SYSTEM Scenario_1
  (* Version 1.0, 2025-08-19, DEVIASH *)
  APPLICATION Scenario_1App (* VDMA *)
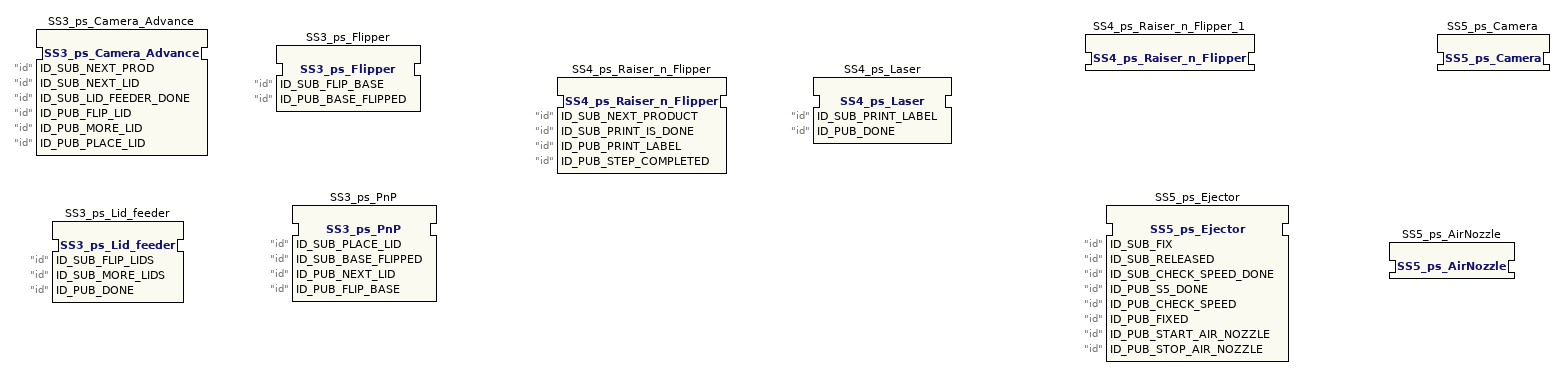
    (* Group S3_Capping_Station: Puting cap on the spinner *)
    (* Group S4_Laser_Print: Printing label on spinner using Laser *)
    (* Group S5_Quality: Speed and label quality check *)
    FBS
      SS3_ps_PnP : SS3_ps_PnP(ID_SUB_PLACE_LID := "id", ID_SUB_BASE_FLIPPED := "id", ID_PUB_NEXT_LID := "id", ID_PUB_FLIP_BASE := "id"); {SET_ATTRIBUTE(GroupName, S3_Capping_Station)}
      SS3_ps_Flipper : SS3_ps_Flipper(ID_SUB_FLIP_BASE := "id", ID_PUB_BASE_FLIPPED := "id"); {SET_ATTRIBUTE(GroupName, S3_Capping_Station)}
      SS3_ps_Lid_feeder : SS3_ps_Lid_feeder(ID_SUB_FLIP_LIDS := "id", ID_SUB_MORE_LIDS := "id", ID_PUB_DONE := "id"); {SET_ATTRIBUTE(GroupName, S3_Capping_Station)}
      SS3_ps_Camera_Advance : SS3_ps_Camera_Advance(ID_SUB_NEXT_PROD := "id", ID_SUB_NEXT_LID := "id", ID_SUB_LID_FEEDER_DONE := "id", ID_PUB_FLIP_LID := "id", ID_PUB_MORE_LID := "id", ID_PUB_PLACE_LID := "id"); {SET_ATTRIBUTE(GroupName, S3_Capping_Station)}
      SS4_ps_Raiser_n_Flipper : SS4_ps_Raiser_n_Flipper(ID_SUB_NEXT_PRODUCT := "id", ID_SUB_PRINT_IS_DONE := "id", ID_PUB_PRINT_LABEL := "id", ID_PUB_STEP_COMPLETED := "id"); {SET_ATTRIBUTE(GroupName, S4_Laser_Print)}
      SS4_ps_Laser : SS4_ps_Laser(ID_SUB_PRINT_LABEL := "id", ID_PUB_DONE := "id"); {SET_ATTRIBUTE(GroupName, S4_Laser_Print)}
      SS5_ps_Ejector : SS5_ps_Ejector(ID_SUB_FIX := "id", ID_SUB_RELEASED := "id", ID_SUB_CHECK_SPEED_DONE := "id", ID_PUB_S5_DONE := "id", ID_PUB_CHECK_SPEED := "id", ID_PUB_FIXED := "id", ID_PUB_START_AIR_NOZZLE := "id", ID_PUB_STOP_AIR_NOZZLE := "id"); {SET_ATTRIBUTE(GroupName, S5_Quality)}
      SS5_ps_AirNozzle : SS5_ps_AirNozzle; {SET_ATTRIBUTE(GroupName, S5_Quality)}
      SS4_ps_Raiser_n_Flipper_1 : SS4_ps_Raiser_n_Flipper; {SET_ATTRIBUTE(GroupName, S5_Quality)}
      SS5_ps_Camera : SS5_ps_Camera; {SET_ATTRIBUTE(GroupName, S5_Quality)}
    END_FBS
  END_APPLICATION
  APPLICATION Scenario_1_with_split_S5App
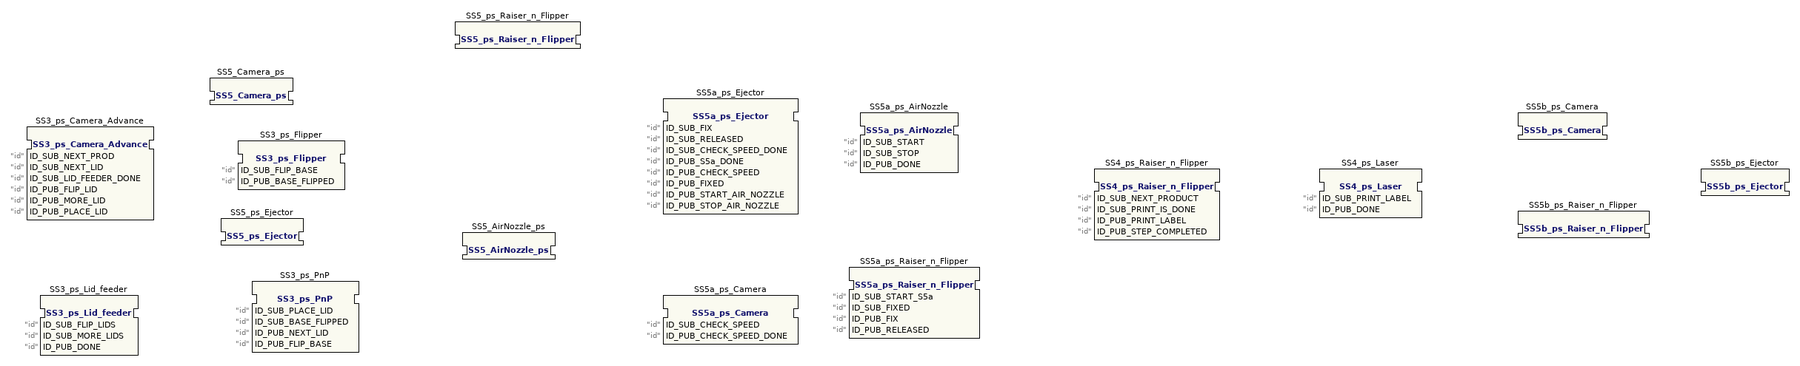
    (* Group S4_Laser_Print: Printing label on spinner using Laser *)
    (* Group S3_Capping_Station: Puting cap on the spinner *)
    (* Group S5a: Speed Quality Check *)
    (* Group S5b: Label Quality Check *)
    FBS
      SS4_ps_Raiser_n_Flipper : SS4_ps_Raiser_n_Flipper(ID_SUB_NEXT_PRODUCT := "id", ID_SUB_PRINT_IS_DONE := "id", ID_PUB_PRINT_LABEL := "id", ID_PUB_STEP_COMPLETED := "id"); {SET_ATTRIBUTE(GroupName, S4_Laser_Print)}
      SS4_ps_Laser : SS4_ps_Laser(ID_SUB_PRINT_LABEL := "id", ID_PUB_DONE := "id"); {SET_ATTRIBUTE(GroupName, S4_Laser_Print)}
      SS3_ps_PnP : SS3_ps_PnP(ID_SUB_PLACE_LID := "id", ID_SUB_BASE_FLIPPED := "id", ID_PUB_NEXT_LID := "id", ID_PUB_FLIP_BASE := "id"); {SET_ATTRIBUTE(GroupName, S3_Capping_Station)}
      SS3_ps_Flipper : SS3_ps_Flipper(ID_SUB_FLIP_BASE := "id", ID_PUB_BASE_FLIPPED := "id"); {SET_ATTRIBUTE(GroupName, S3_Capping_Station)}
      SS3_ps_Lid_feeder : SS3_ps_Lid_feeder(ID_SUB_FLIP_LIDS := "id", ID_SUB_MORE_LIDS := "id", ID_PUB_DONE := "id"); {SET_ATTRIBUTE(GroupName, S3_Capping_Station)}
      SS3_ps_Camera_Advance : SS3_ps_Camera_Advance(ID_SUB_NEXT_PROD := "id", ID_SUB_NEXT_LID := "id", ID_SUB_LID_FEEDER_DONE := "id", ID_PUB_FLIP_LID := "id", ID_PUB_MORE_LID := "id", ID_PUB_PLACE_LID := "id"); {SET_ATTRIBUTE(GroupName, S3_Capping_Station)}
      SS5_AirNozzle_ps : SS5_AirNozzle_ps; {SET_ATTRIBUTE(GroupName, S5_Quality)}
      SS5_Camera_ps : SS5_Camera_ps; {SET_ATTRIBUTE(GroupName, S5_Quality)}
      SS5_ps_Ejector : SS5_ps_Ejector; {SET_ATTRIBUTE(GroupName, S5_Quality)}
      SS5_ps_Raiser_n_Flipper : SS5_ps_Raiser_n_Flipper; {SET_ATTRIBUTE(GroupName, S5_Quality)}
      SS5a_ps_AirNozzle : SS5a_ps_AirNozzle(ID_SUB_START := "id", ID_SUB_STOP := "id", ID_PUB_DONE := "id"); {SET_ATTRIBUTE(GroupName, S5a)}
      SS5a_ps_Camera : SS5a_ps_Camera(ID_SUB_CHECK_SPEED := "id", ID_PUB_CHECK_SPEED_DONE := "id"); {SET_ATTRIBUTE(GroupName, S5a)}
      SS5a_ps_Ejector : SS5a_ps_Ejector(ID_SUB_FIX := "id", ID_SUB_RELEASED := "id", ID_SUB_CHECK_SPEED_DONE := "id", ID_PUB_S5a_DONE := "id", ID_PUB_CHECK_SPEED := "id", ID_PUB_FIXED := "id", ID_PUB_START_AIR_NOZZLE := "id", ID_PUB_STOP_AIR_NOZZLE := "id"); {SET_ATTRIBUTE(GroupName, S5a)}
      SS5b_ps_Camera : SS5b_ps_Camera; {SET_ATTRIBUTE(GroupName, S5b)}
      SS5b_ps_Ejector : SS5b_ps_Ejector; {SET_ATTRIBUTE(GroupName, S5b)}
      SS5b_ps_Raiser_n_Flipper : SS5b_ps_Raiser_n_Flipper; {SET_ATTRIBUTE(GroupName, S5b)}
      SS5a_ps_Raiser_n_Flipper : SS5a_ps_Raiser_n_Flipper(ID_SUB_START_S5a := "id", ID_SUB_FIXED := "id", ID_PUB_FIX := "id", ID_PUB_RELEASED := "id"); {SET_ATTRIBUTE(GroupName, S5a)}
    END_FBS
  END_APPLICATION
  APPLICATION Scenario_1_baseline_S5
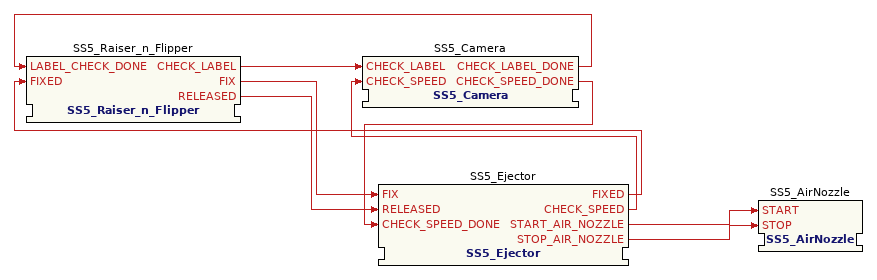
    FBS
      SS5_AirNozzle : SS5_AirNozzle;
      SS5_Camera : SS5_Camera;
      SS5_Ejector : SS5_Ejector;
      SS5_Raiser_n_Flipper : SS5_Raiser_n_Flipper;
    END_FBS
    EVENT_CONNECTIONS
      SS5_Raiser_n_Flipper.CHECK_LABEL TO SS5_Camera.CHECK_LABEL;
      SS5_Camera.CHECK_LABEL_DONE TO SS5_Raiser_n_Flipper.LABEL_CHECK_DONE;
      SS5_Raiser_n_Flipper.FIX TO SS5_Ejector.FIX;
      SS5_Ejector.FIXED TO SS5_Raiser_n_Flipper.FIXED;
      SS5_Raiser_n_Flipper.RELEASED TO SS5_Ejector.RELEASED;
      SS5_Ejector.CHECK_SPEED TO SS5_Camera.CHECK_SPEED;
      SS5_Ejector.START_AIR_NOZZLE TO SS5_AirNozzle.START;
      SS5_Ejector.STOP_AIR_NOZZLE TO SS5_AirNozzle.STOP;
      SS5_Camera.CHECK_SPEED_DONE TO SS5_Ejector.CHECK_SPEED_DONE;
    END_CONNECTIONS
  END_APPLICATION
  APPLICATION Scenario_1_baseline_Sa_S5b
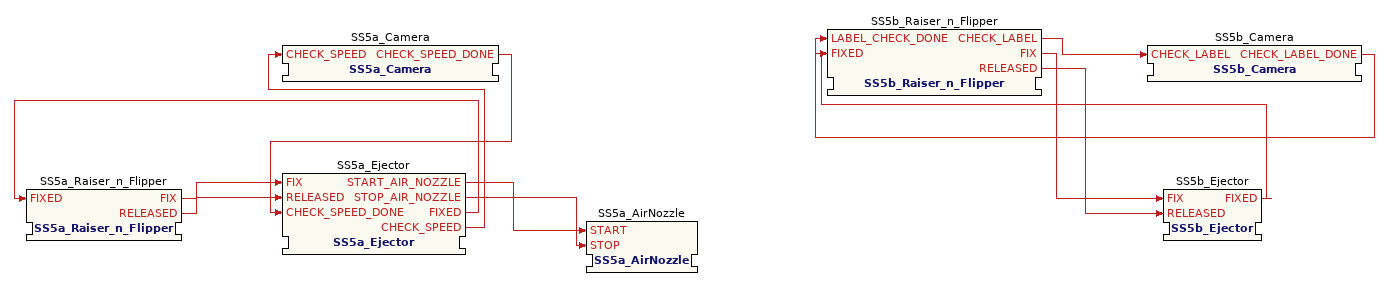
    FBS
      SS5a_AirNozzle : SS5a_AirNozzle;
      SS5a_Camera : SS5a_Camera;
      SS5a_Ejector : SS5a_Ejector;
      SS5a_Raiser_n_Flipper : SS5a_Raiser_n_Flipper;
      SS5b_Camera : SS5b_Camera;
      SS5b_Ejector : SS5b_Ejector;
      SS5b_Raiser_n_Flipper : SS5b_Raiser_n_Flipper;
    END_FBS
    EVENT_CONNECTIONS
      SS5b_Raiser_n_Flipper.CHECK_LABEL TO SS5b_Camera.CHECK_LABEL;
      SS5b_Camera.CHECK_LABEL_DONE TO SS5b_Raiser_n_Flipper.LABEL_CHECK_DONE;
      SS5b_Raiser_n_Flipper.FIX TO SS5b_Ejector.FIX;
      SS5b_Ejector.FIXED TO SS5b_Raiser_n_Flipper.FIXED;
      SS5b_Raiser_n_Flipper.RELEASED TO SS5b_Ejector.RELEASED;
      SS5a_Ejector.START_AIR_NOZZLE TO SS5a_AirNozzle.START;
      SS5a_Ejector.STOP_AIR_NOZZLE TO SS5a_AirNozzle.STOP;
      SS5a_Ejector.FIXED TO SS5a_Raiser_n_Flipper.FIXED;
      SS5a_Raiser_n_Flipper.FIX TO SS5a_Ejector.FIX;
      SS5a_Raiser_n_Flipper.RELEASED TO SS5a_Ejector.RELEASED;
      SS5a_Ejector.CHECK_SPEED TO SS5a_Camera.CHECK_SPEED;
      SS5a_Camera.CHECK_SPEED_DONE TO SS5a_Ejector.CHECK_SPEED_DONE;
    END_CONNECTIONS
  END_APPLICATION
END_SYSTEM
